// TIA Portal V18 export
// export: Created 2026-06-20T13:30:08.4779411Z, ExportSetting WithDefaults, DisplayName Totally Integrated Automation Portal, DisplayVersion V18, DisplayName TIA Portal Openness, DisplayVersion V18, DisplayName TIA Portal Version Control Interface, DisplayVersion V18, DisplayName STEP 7 Professional, DisplayVersion V18, DisplayName STEP 7 Safety, DisplayVersion V18, DisplayName WinCC Professional, DisplayVersion V18
DATA_BLOCK "Timers_PLC1"   // DB1
TITLE = Timers_PLC1
{ S7_Optimized_Access := 'TRUE' }
VERSION : 0.1
// Global DB containing all timers and PID instances
// stored: AutoNumber true, DBAccessibleFromOPCUA true, IsOnlyStoredInLoadMemory false, IsRetainMemResEnabled false, IsWriteProtectedInAS false, MemoryReserve 100
   VAR
      Timer_Dosing_Bon1 : IEC_TIMER;
      Timer_Tip_Bon1 : IEC_TIMER;
      Timer_Dosing_Bon2 : IEC_TIMER;
      Timer_Tip_Bon2 : IEC_TIMER;
      Timer_Khuay_Bon1 : IEC_TIMER;
      Timer_Khuay_Thuan_Bon2 : IEC_TIMER;
      Timer_Khuay_Nghich_Bon2 : IEC_TIMER;
      Timer_Thanh_Trung_Bon2 : IEC_TIMER;
      Timer_DryRun_Bon2 : IEC_TIMER;
      Timer_Heartbeat_PLC1 : IEC_TIMER;
      VFD_Bon2_MB_Counter : IEC_COUNTER;
   END_VAR
BEGIN
END_DATA_BLOCK
